(* IEC 61131-3 sources: CodesysTest/export/SX.dev/Plc Logic/Application/HMIData, 3 files *)

(* ---- HMI.gvl.st ---- *)
(*#-#-#-#-#-#-#-#-#-#---Declaration---#-#-#-#-#-#-#-#-#-#-#-#-#*)

{attribute 'qualified_only'}
{attribute 'global_init_slot' := '50001'}
VAR_GLOBAL
	data : FB_HMIDataSX;
END_VAR

(* ---- HMIData.gvl.st ---- *)
(*#-#-#-#-#-#-#-#-#-#---Declaration---#-#-#-#-#-#-#-#-#-#-#-#-#*)

{attribute 'qualified_only'}
{attribute 'global_init_slot' := '50001'}
VAR_GLOBAL
	initiateCycle : BOOL;  // Initiate Cycle Pushbutton
	ackAllFaults : BOOL; // Acknowledge All Faults from HMI
	makeReady : BOOL;
	homeMachine : BOOL;
	machineHomed : BOOL;
	pressureBarState : STRING;
	activeScreen : DINT;
	jawService : ServiceCommands;
	jawJogOpen : BOOL;
	jawjobClosed : BOOL;
	loadPlateService : ServiceCommands;
	IBDService : ServiceCommands;
	IBDJogOpen : BOOL;
	IBDJogClosed : BOOL;
	jogFilmForward : BOOL;
	jogFilmReverse : BOOL;
	cycleSealer : BOOL;
	printHeadService : ServiceCommands;
	startJawCycleTest : BOOL;
	stopJawCycleTest : BOOL;
	jawCycleTestCycles : DINT;
	jawCycleTestActive : BOOL;
	teachBagPhotoeye : BOOL;
	teachingBagPhoteye : BOOL;
	factoryHomeJaw : BOOL;
    stopMachine : BOOL;
	inCycle : BOOL;
	resetAverageCycleTime : BOOL;
	profaceInterface : ARRAY[0..20] OF INT;
	bannerMessageIndication : DINT;
	faultActive : BOOL;
	simulateAllIO : BOOL;
	activeFaults : ARRAY[0..GlobalObjects.MAX_FAULTS] OF STRING;
	passthroughActual : REAL;
	currentPackMLState : STRING;
	BPMBagsMade : UDINT;
	BPMActiveTime : STRING;
	BPMBagsPerMinute : REAL;
	BPMReset : BOOL;
	cycleTime : REAL;
	printerReady : BOOL;
	bagDeliveryReady : BOOL;
	loadPlateReady : BOOL;
	jawReady : BOOL;
	bcvReady : BOOL;
	IBDReady : BOOL;
	sendSampleLabels : BOOL;
	clearAllLabels : BOOL;
	printerAndVerifierEnablePB : BOOL;
	printerAndVerifierEnableIndication : BOOL;
	frontJawMotorData : sctOrientalHMIData;
	rearJawMotorData : sctOrientalHMIData;
	loadPlateMotorData : sctOrientalHMIData;
	IBDMotorData : sctOrientalHMIData;
	bagDeliveryMotorData : sctAppliedMotionHMIData;
	barcodeReadGoodIndication : BOOL;
	barcodeReadBadIndication : BOOL;
	barcodeVerifierTrigger : BOOL;
END_VAR

VAR_GLOBAL PERSISTENT RETAIN
	bagsMade : UDINT;
	batchEnable : BOOL;
	batchSetting : UDINT := 10;
	batchCount : UDINT;
	headCycleCount : UDINT;
	pressureBarOpenDelay : REAL;
	pressureBarCloseDelay : REAL;
	passthroughSetting : REAL := 5.5;
	sealBarDwell : REAL := 0.2;
	sealBarCool : REAL := 0.4;
	bagSkirtLength : REAL := 2;
	bagLength : REAL := 17.62;
	bagWidth : REAL := 11;
	bagThickness : REAL := 2.5;
	bagForwardSpeed : UDINT := 40;
	bagReverseSpeed : UDINT := 8;
	printSpeed : UDINT := 6;
	printLength : REAL := 1.25;
	printOffset : REAL := 10.0;
	fillerCountSetting : UDINT;
	fillerCurrentCount : UDINT;
	fillerDropTime : REAL;
	loadPlateDelay : REAL;
	loadPlateDwell : REAL := 0.1;
	IBDInUse : BOOL := TRUE;
	IBDInstalled : BOOL := TRUE;
	IBDOpenMotionProfile : sctMotionProfile := (velo := 9.0, accel := 30.0, decel := 50.0, current := 100.0);
	IBDCloseMotionProfile : sctMotionProfile := (velo := 15.0, accel := 10.0, decel := 10.0, current := 50.0);
	IBDZeroOffset : REAL := 2.0;
	jawCloseDelay : REAL := 0.1;
	jawClosePositionSetting : REAL := -0.45;
	jawOpenMotionProfile : sctMotionProfile := (velo := 14.0, accel := 300.0, decel := 300.0, current := 100.0);
	jawCloseMotionProfile : sctMotionProfile := (velo := 14.0, accel := 10.0, decel := 10.0, current := 100.0);
	jawZeroOffset : REAL := 2.0;
	lastCycleTime : REAL;
	bagDropClearanceDwell : REAL := 0.5;
	averageCycleTime : REAL;
	currentJobID : INT;
	separateBeforeSeal : BOOL := TRUE;
	partsCounterEnable : BOOL;
	partsCounterCount : UDINT;
	partsCounterSetting : UDINT;
	consecutiveBagsEnable : BOOL;
	consecutiveBagsCount : UDINT;
	consecutiveBagsSetting : UDINT;
	printerInstalled : BOOL := TRUE;
	printerInUse : BOOL := TRUE;
	printerCancelRequest : BOOL;
	barcodeVerifierInstalled : BOOL := TRUE;
	barcodeGoodReadCount : UDINT;
	barcodeBadReadCount : UDINT;
	barcodeBadReadFaultSetting : UDINT := 1;
	barcodeStartPosition : REAL := 3.0;
	barcodeScanDistance : REAL := 0.1;
	barcodeVerifierInUse : BOOL := TRUE;
	loadPlateInstalled : BOOL := TRUE;
	loadPlateLoweredPositionSetting : REAL := 0;
	loadPlateRaisedPositionSetting :  REAL := 1;
	loadPlateInUse : BOOL := TRUE;
	loadPlateRaiseProfile : sctMotionProfile := (velo := 3.0, accel := 100.0, decel := 10.0, current := 100.0);
	loadPlateLowerProfile : sctMotionProfile := (velo := 5.0, accel := 100.0, decel := 100.0, current := 100.0);
	fillerEnable : BOOL;
	autoModeEnable : BOOL;
	autoModeDwell : REAL;
	dryCycleEnable : BOOL;
END_VAR

VAR_GLOBAL CONSTANT
	version : STRING := '1.0.7.1';
END_VAR

(* ---- FB_HMIDataSX.pou.st ---- *)
(*#-#-#-#-#-#-#-#-#-#---Declaration---#-#-#-#-#-#-#-#-#-#-#-#-#*)

{attribute 'FBVisuCreator'}
FUNCTION_BLOCK FB_HMIDataSX
VAR_INPUT
	initiateCycle : BOOL;  // Initiate Cycle Pushbutton
	ackAllFaults : BOOL; // Acknowledge All Faults from HMI
	makeReady : BOOL;
	jawService : ServiceCommands;
	jawJogOpen : BOOL;
	jawjobClosed : BOOL;
	loadPlateService : ServiceCommands;
	IBDService : ServiceCommands;
	IBDJogOpen : BOOL;
	IBDJogClosed : BOOL;
	jogFilmForward : BOOL;
	jobFilmReverse : BOOL;
	homeMachine : BOOL;
	machineHomed : BOOL;
	cycleSealer : BOOL;
	printHeadService : ServiceCommands;
	startJawCycleTest : BOOL;
	stopJawCycleTest : BOOL;
	jawCycleTestCount : FB_MachineCounter(name := 'Jaw Cycle Test Counter');
	teachBagPhotoeye : BOOL;
	teachingBagPhoteye : BOOL;
	factoryHomeJaw : BOOL;
    stopMachine : BOOL;
	printerAndVerifierEnablePB : BOOL;
	printerAndVerifierEnableIndication : BOOL;
	BPMBagsMade : DINT;
	BPMActiveTime : REAL;
	BPMBagsPerMinute : REAL;
	BPMReset : BOOL;
	{attribute 'FBVisuCreatorFormatString' := '%s'}
	version : STRING := '0.2A';
	inCycle : BOOL;
	batchEnable : BOOL;
	{attribute 'FBVisuCreatorFormatString' := '%d'}
	batchSetting : UDINT := 10;
	{attribute 'FBVisuCreatorFormatString' := '%d'}
	batchCount : UDINT;
	{attribute 'FBVisuCreatorFormatString' := '%d'}
	headCycleCount : UDINT;
	{attribute 'FBVisuCreatorFormatString' := '%1.2f'}
	pressureBarOpenDelay : REAL;
	{attribute 'FBVisuCreatorFormatString' := '%1.2f'}
	pressureBarCloseDelay : REAL;
	{attribute 'FBVisuCreatorFormatString' := '%1.2f'}
	passthroughSetting : REAL := 8.0;
	{attribute 'FBVisuCreatorFormatString' := '%1.2f'}
	passthroughActual : REAL;
	{attribute 'FBVisuCreatorFormatString' := '%1.2f'}
	lpaDwell : REAL;
	{attribute 'FBVisuCreatorFormatString' := '%1.2f'}
	hpaDwell : REAL;
	{attribute 'FBVisuCreatorFormatString' := '%1.2f'}
	sealBarDwell : REAL := 0.0;
	{attribute 'FBVisuCreatorFormatString' := '%1.2f'}
	sealBarCool : REAL := 0.0;
	{attribute 'FBVisuCreatorFormatString' := '%d'}
	sealBarTemperatureSetting : UDINT;
	{attribute 'FBVisuCreatorFormatString' := '%d'}
	sealBarTemperature : UDINT;
	{attribute 'FBVisuCreatorFormatString' := '%1.2f'}
	sealFlattenerBagOpenPositionSetting : REAL;
	{attribute 'FBVisuCreatorFormatString' := '%1.2f'}
	sealFlattenerFlattenedPositionSetting : REAL;
	{attribute 'FBVisuCreatorFormatString' := '%1.2f'}
	sealFlattenerMoveInPositionSetting : REAL;
	{attribute 'FBVisuCreatorFormatString' := '%1.2f'}
	bagSkirtLength : REAL := 1.35;
	{attribute 'FBVisuCreatorFormatString' := '%1.2f'}
	bagLength : REAL := 23.5;
	{attribute 'FBVisuCreatorFormatString' := '%1.2f'}
	bagWidth : REAL := 17.5;
	{attribute 'FBVisuCreatorFormatString' := '%1.2f'}
	bagThickness : REAL := 2.5;
	{attribute 'FBVisuCreatorFormatString' := '%d'}
	bagForwardSpeed : UDINT := 55;
	{attribute 'FBVisuCreatorFormatString' := '%d'}
	bagReverseSpeed : UDINT := 3;
	{attribute 'FBVisuCreatorFormatString' := '%d'}
	printSpeed : UDINT := 6;
	{attribute 'FBVisuCreatorFormatString' := '%1.2f'}
	printLength : REAL := 8.0;
	{attribute 'FBVisuCreatorFormatString' := '%1.2f'}
	printOffset : REAL := 2.0;
	{attribute 'FBVisuCreatorFormatString' := '%d'}
	fillerCountSetting : UDINT;
	{attribute 'FBVisuCreatorFormatString' := '%d'}
	fillerCurrentCount : UDINT;
	{attribute 'FBVisuCreatorFormatString' := '%1.2f'}
	fillerDropTime : REAL;
	{attribute 'FBVisuCreatorFormatString' := '%1.2f'}
	loadPlateDelay : REAL;
	{attribute 'FBVisuCreatorFormatString' := '%1.2f'}
	loadPlateDwell : REAL := 2.5;
	IBDInUse : BOOL;
	IBDInstalled : BOOL;
	IBDCurrentSetting : REAL := 50.0;
	jawCloseDelay : REAL := 0.2;
	jawClosePositionSetting : REAL := -0.2;
	exitConveyorService: ServiceCommands;
	{attribute 'FBVisuCreatorFormatString' := '%1.2f'}
	exitConveyorDwell : REAL := 9.0;
	{attribute 'FBVisuCreatorFormatString' := '%1.2f'}
	lastCycleTime : REAL;
	{attribute 'FBVisuCreatorFormatString' := '%1.2f'}
	bagDropClearanceDwell : REAL := 0.5;
	{attribute 'FBVisuCreatorFormatString' := '%1.2f'}
	averageCycleTime : REAL;
	resetAverageCycleTime : BOOL;
	{attribute 'FBVisuCreatorFormatString' := '%d'}
	bagOpenRetrySetting : UINT := 3;
	{attribute 'FBVisuCreatorFormatString' := '%d'}
	bagOpenRetryCount : UINT;
	{attribute 'FBVisuCreatorFormatString' := '%d'}
	currentJobID : INT;
	separateBeforeSeal : BOOL := TRUE;
	activateDemoMode : BOOL;
	bagOpenAssistEnable : BOOL := TRUE;
	bagOpenSensorEnable : BOOL := TRUE;
	{attribute 'FBVisuCreatorFormatString' := '%1.2f'}
	grabBagDelay : REAL := 0.5;
	{attribute 'FBVisuCreatorFormatString' := '%1.2f'}
	checkForBagOpenDelay : REAL := 1.0;
	{attribute 'FBVisuCreatorFormatString' := '%1.2f'}
	bagClearedFromFingersDelay : REAL := 0.5;
	{attribute 'FBVisuCreatorFormatString' := '%1.2f'}
	vacuumDwell : REAL := 0.5;
	(*Faults*)
	{attribute 'FBVisuCreatorFormatString' := '%s'}
	pressureBarState : STRING;
	activeScreen : DINT;
	profaceInterface : ARRAY[0..20] OF INT;
	partsCounterEnable : BOOL;
	partsCounterCount : UDINT;
	partsCounterSetting : UDINT;
	consecutiveBagsEnable : BOOL;
	consecutiveBagsCount : UDINT;
	consecutiveBagsSetting : UDINT;
	printerInstalled : BOOL;
	printerInUse : BOOL;
	printerCancelRequest : BOOL;
	barcodeVerifierInstalled : BOOL;
	barcodeGoodReadCount : UDINT;
	barcodeBadReadCount : UDINT;
	barcodeBadReadFaultSetting : UDINT;
	barcodeStartPosition : REAL;
	barcodeScanDistance : REAL := 1.0;
	barcodeVerifierInUse : BOOL;
	barcodeLastReadString : STRING[100];
	barcodeReadGoodIndication : BOOL;
	barcodeReadBadIndication : BOOL;
	loadPlateInstalled : BOOL;
	loadPlateInUse : BOOL;
	fillerEnable : BOOL;
	autoModeEnable : BOOL;
	autoModeDwell : REAL := 0.75;
	bannerManager : FB_BannerManager;
    (*Counters*)
    baggerCycles : FB_MachineCounter(name := 'Bagger Cycle Counter');
	pressureBarCycles : FB_MachineCounter(name := 'Pressure Bar Cycle Counter');
	//passthroughChanges : FB_MachineCounter(name := 'Passthrough Changes Counter');
	//loadPlateCycles : FB_MachineCounter(name := 'Load Plate Cycle Counter');
	//printerCycles : FB_MachineCounter(name := 'Printer Cycle Counter');
	//motorizedSealFlattenerCycles : FB_MachineCounter(name := 'Motorized Seal Flattener Cycles');
	//bagOpenRetryTotal : FB_MachineCounter(name := 'Bag Open Retry Totals');
	(*Info*)
	faultActive : BOOL;
	simulateAllIO : BOOL;
	(*
	(*Factoy Config*)
	bofSelection : BagOpenFingersSelection := BagOpenFingersSelection.PneumaticWithBagOpenSensors;
	bofEnable : BOOL := TRUE;
	sealFlattenersSelection : SealFlattenerSelection := SealFlattenerSelection.MotorizedSealFlatteners;
	sealFlattenersEnable : BOOL := TRUE;
	printerSelection : LabelPrinterSelection := LabelPrinterSelection.ZebraPrinter;
	printerEnable : BOOL := TRUE;
	integratedExitConveyorSelection : IntegratedConveyorSelection := IntegratedConveyorSelection.RearExit;
	integratedExitConveyorEnable : BOOL := TRUE;
	packageEjectSelection : PackageEjectionSelection := PackageEjectionSelection.RearRetractingLoadPlate;
	packageEjectEnable : BOOL := TRUE;
	*)

	(*I/O*)

END_VAR
VAR_OUTPUT
END_VAR
VAR
END_VAR
(*#-#-#-#-#-#-#-#-#-#---Implementation---#-#-#-#-#-#-#-#-#-#-#-#-#*)
